// TIA Portal V19 export
VAR_GLOBAL   // PLC tag table "Prod_Err_Code_CONST"
END_VAR
VAR_GLOBAL CONSTANT   // user constants
   PROD_ERR_Type_UNKNOW : DInt := -101;   // Prod_Item.Type - Valore errato
   PROD_ERR_O_ID_empty : DInt := -102;   // Prod.item.O_ID - Vuoto
   PROD_ERR_MES_IDP_Empty : DInt := -103;   // Prod_item.MES_IDP - Vuoto e ordine caricato dal MES (Prod_Item.Type = 1)
   PROD_ERR_MES_IDP_NOT_Empty : DInt := -104;   // Prod_item.MES_IDP - NON Vuoto e ordine caricato dal HMI (Prod_Item.Type = 2)
   PROD_ERR_PPrfNo_Empty : DInt := -105;   // Prod_item.PPrfNo <= 0 - il numero del programma profilo è <= 0
   PROD_ERR_PPrfNo_NotExist : DInt := -106;   // Prod_item.PPrfNo > 0 ma il numero del programma profilo NON esiste nella lista PIVOT dei programmi ("PPrf_MAIN".PIVOT)
   PROD_ERR_PPrf_Name_Mismatch : DInt := -107;
   PROD_ERR_Beam_W_A_Min : DInt := -108;
   PROD_ERR_Beam_W_A_Max : DInt := -109;
   PROD_ERR_Beam_H_B_Min : DInt := -110;
   PROD_ERR_Beam_H_B_Max : DInt := -111;
   PROD_ERR_Beam_Tickness_Min : DInt := -112;
   PROD_ERR_Beam_Tickness_Max : DInt := -113;
   PROD_ERR_Beams_REQ_empty : DInt := -114;
   PROD_ERR_Parts_REQ_empty : DInt := -115;
   PROD_ERR_Len_min : DInt := -116;
   PROD_ERR_Len_max : DInt := -117;
   PROD_ERR_No_Parts_ToGo : DInt := -118;
   PROD_ERR_PPrf_MISMATCH_PPrf_LINE_SETUP : DInt := -201;
   PROD_ERR_PPrf_MIISMATCH_PPrf_ON_WORK : DInt := -202;
   PROD_ERR_O_ACT_FULL : DInt := -301;
   PROD_ERR_O_TODO_INDEX_EXCEEDS_BOUNDS : DInt := -302;   // L'indice di selezione ordine su O_TODO è fuori dai limit 1..."PROD_TODO_ITEMS"
   PROD_ERR_O_ENDING_INDEX_EXCEEDS_BOUNDS : DInt := -402;
   PROD_FUN_RESULT_OK : DInt := 0;
   PROD_FUN_RESULT_BUFFER_EMPTY : DInt := 1;
   PROD_FUN_RESULT_CLEAR_GAP_DONE : DInt := 0;
   PROD_FUN_RESULT_NO_GAP : DInt := 2;
   PROD_ERR_PPrf_Get_Error : DInt := -130;
   PROD_ERR_PPrf_Get_Timeout : DInt := -131;
   PROD_ERR_PPRF_MISMATCH_BEAM_TYPE : DInt := -132;
   PROD_ERR_PPRF_MISMATCH_BEAM_W_A : DInt := -133;
   PROD_ERR_PPRF_MISMATCH_BEAM_H_B : DInt := -134;
   PROD_ERR_PPRF_MISMATCH_BEAM_TICKNESS : DInt := -135;
   PROD_ERR_BUFFER_MSGs_SHIFT : DInt := -1004;
   PROD_ERR_ORDER_NOT_FOUND : DInt := -1011;
   PROD_ORDER_IS_AT_O_ACT : DInt := 0;   // L'ordine si trova su "Production".O_ACT = In lavoro con taglio Part in corso
   PROD_ORDER_IS_AT_O_TODO : DInt := 1;   // L'ordine si trova su "Production".O_TODO =Nella coda degli ordini da produrre
   PROD_ORDER_IS_AT_O_ENDING : DInt := 2;   // L'ordine si trova su "Production".O_ENDING = In lavoro con taglio Part concluso ma BEAM non conclusi
   PROD_ORDER_IS_AT_O_OUT : DInt := 3;   // L'ordine si trova su "Production".O_OUT= Fuori dal processo = Ordine concluso
   PROD_ERR_BUFFER_MSGs_FULL : DInt := -1005;
   PROD_ERR_BUFFER_MSGs_INDEX_EXCEEDS_BOUNDS : DInt := -1002;
   PROD_ERR_O_ID_AND_MES_IDP_NOT_VALID : DInt := -1010;   // La funzione "Prod_Item_GetData" non è om grado di cercare l'rdine perchè sia O_ID che MES_IDP sono non valorizzate
   PROD_ERR_BUFFER_MSGs_UNKNOW_TOPIC : DInt := -1000;
   PROD_ERR_CALC_PACK_DIM_X : DInt := -120;   // Errore larghezza pacco va fuori misura
   PROD_ERR_CALC_PACK_DIM_Z : DInt := -121;   // Errore altezza pacco va fuori misura
   ERR_KEY_IDP : DInt := -3000;   // [IDP] Chiave non trovata
   ERR_DEL_IDP : DInt := -3001;   // [IDP] Delimitatore valore non trovato
   ERR_VAL_IDP : DInt := -3002;   // [IDP] Valore nullo
   ERR_KEY_TYP : DInt := -3003;   // [TYP] Chiave non trovata
   ERR_DEL_TYP : DInt := -3004;   // [TYP] Delimitatore valore non trovato
   ERR_VAL_TYP : DInt := -3005;   // [TYP] Valore errato
   ERR_KEY_W : DInt := -3006;   // [W] Chiave non trovata
   ERR_DEL_W : DInt := -3007;   // [W] Delimitatore valore non trovato
   ERR_VAL_NUM_W : DInt := -3008;   // [W] Valore non è un numero
   ERR_KEY_H : DInt := -3009;   // [H] Chiave non trovata
   ERR_DEL_H : DInt := -3010;   // [H] Delimitatore valore non trovato
   ERR_VAL_NUM_H : DInt := -3020;   // [H] Valore non è un numero
   ERR_KEY_TK : DInt := -3021;   // [TK] Chiave non trovata
   ERR_DEL_TK : DInt := -3022;   // [TK] Delimitatore valore non trovato
   ERR_VAL_NUM_TK : DInt := -3023;   // [TK] Valore non è un numero
   ERR_KEY_LN : DInt := -3024;   // [LN] Chiave non trovata
   ERR_DEL_LN : DInt := -3025;   // [LN] Delimitatore valore non trovato
   ERR_VAL_NUM_LN : DInt := -3026;   // [LN] Valore non è un numero
   ERR_KEY_QQ : DInt := -3027;   // [QQ] Chiave non trovata
   ERR_DEL_QQ : DInt := -3028;   // [QQ] Delimitatore valore non trovato
   ERR_VAL_NUM_QQ : DInt := -3029;   // [QQ] Valore non è un numero
   ERR_KEY_RR : DInt := -3030;   // [RR] Chiave non trovata
   ERR_DEL_RR : DInt := -3031;   // [RR] Delimitatore valore non trovato
   ERR_VAL_NUM_RR : DInt := -3032;   // [RR] Valore non è un numero
   ERR_KEY_DC : DInt := -3033;   // [DC] Chiave non trovata
   ERR_DEL_DC : DInt := -3034;   // [DC] Delimitatore valore non trovato
   ERR_VAL_NUM_DC : DInt := -3035;   // [DC] Valore errato
   ERR_KEY_DE : DInt := -3036;   // [DC] Chiave non trovata
   ERR_DEL_DE : DInt := -3037;   // [DC] Delimitatore valore non trovato
   ERR_VAL_NUM_DE : DInt := -3038;   // [DC] Valore errato
   ERR_KEY_KA : DInt := -3039;   // [KA] Chiave non trovata
   ERR_DEL_KA : DInt := -3040;   // [KA] Delimitatore valore non trovato
   ERR_VAL_NUM_KA : DInt := -3041;   // [KA] Valore errato
   ERR_KEY_NPR : DInt := -3042;   // [NPR] Chiave non trovata
   ERR_DEL_NPR : DInt := -3043;   // [NPR] Delimitatore valore non trovato
   ERR_VAL_NUM_NPR : DInt := -3044;   // [NPR] Valore errato
   ERR_KEY_NPL : DInt := -3045;   // [NPL] Chiave non trovata
   ERR_DEL_NPL : DInt := -3046;   // [NPL] Delimitatore valore non trovato
   ERR_VAL_NUM_NPL : DInt := -3047;   // [NPR] Valore errato
   ERR_O_CAN_NOT_BE_DELETED_BTRK_PRESENCE : DInt := -3105;   // L'ordine non può essere cancellato perchè ci sono ancora pezzi che lo usano nei B_TRK
   PROD_ERR_BUFFER_ORDERs_FULL : DInt := -2005;
   PROD_ERR_BUFFER_ORDERs_SHIFT : DInt := -2004;
   PROD_ERR_BUFFER_ORDERs_INDEX_EXCEEDS_BOUNDS : DInt := -2002;
   PROD_ERR_BUFFER_ORDERs_NO_SPACE : DInt := -2006;
   PROD_ERR_BTRK_A304_EMPTY : DInt := -1100;   // Errore non ci sono pezzi nella navetta di scarico
   PROD_ERR_MES_IDP_Duplicate : DInt := -119;
   ERR_O_CAN_NOT_BE_DELETED_PTRK_PRESENCE : DInt := -3104;   // L'ordine non può essere cancellato perchè ci sono ancora pezzi che lo usano nei P_TRK
   ERR_O_CAN_NOT_BE_DELETED_IS_O_ACT : DInt := -3101;   // L'ordine non può essere cancellato perchè è in lavoro
   ERR_O_CAN_NOT_BE_DELETED_IS_O_OUT : DInt := -3103;   // L'ordine non può essere cancellato perchè è tra quelli già usciti
   ERR_O_CAN_NOT_BE_DELETED_NOT_PRESENT : DInt := -3100;   // L'ordine non può essere cancellato perchè non è stato trovato
   ERR_O_CAN_NOT_BE_DELETED_IS_O_ENDING : DInt := -3102;   // L'ordine non può essere cancellato perchè è tra quelli in via di completamento
   ERR_SET_UP_MAN_NOT_COMPLETE : DInt := -4000;   // !! TODO nuovo da aggiungere del decoder stringhe
   ERR_KEY_CN : DInt := -3050;
   ERR_DEL_CN : DInt := -3051;
   ERR_VAL_CN : DInt := -3052;
   ERR_KEY_HN : DInt := -3053;
   ERR_DEL_HN : DInt := -3054;
   ERR_VAL_HN : DInt := -3055;
   ERR_KEY_PR : DInt := -3056;
   ERR_DEL_PR : DInt := -3057;
   ERR_VAL_PR : DInt := -3058;
   ERR_COIL_DATA_CAN_NOT_WRITE_ALREADY_PRESENT : DInt := -5000;   // I dati del coil non possono essere scritti perchè già presenti (NO sovrascrittura possibile)
   ERR_COIL_DATA_CAN_NOT_DELETE_DECOILER_NOT_IN_LOAD_POSITION : DInt := -5010;   // I dati coil non possono essere cancellati perchè non è chiaro quale rotolo è in carico
   ERR_COIL_DATA_CAN_NOT_DELETE_DATA_NOT_MATCH : DInt := -5011;   // I dati coil non possono essere cancellati perchè i dati non corrispondono
   ERR_COIL_DATA_CAN_NOT_INC_PROVINO_DATA_NOT_MATCH : DInt := -5030;   // Numero provini non può essere Incrementato perchè i dati non corrispondono
   ERR_COIL_DATA_CAN_NOT_WRITE_DECOILER_NOT_IN_LOAD_POSITION : DInt := -5002;   // I dati del coil non possono essere scritti perchè non consistenti (Numero colata / Numero rotolo non valorizzati)
   PROD_FUN_RESULT_COIL_AT_DECOILER_IN_LINE : DInt := 1;
   PROD_FUN_RESULT_COIL_AT_DECOILER_IN_LOAD : DInt := 2;
END_VAR
